// TIA Portal V15.1 export
// export: Created 2024-06-21T08:40:57.9475663Z, ExportSetting WithDefaults, DisplayName Totally Integrated Automation Portal, DisplayVersion V15.1 Update 5, DisplayName TIA Portal Openness, DisplayVersion V15.1 Update 5, DisplayName SINAMICS Startdrive Advanced, DisplayVersion V15.1, DisplayName G130, G150, S120, S150, SINAMICS MV, S210, DisplayVersion V15.1, DisplayName G110M, G120, G120C, G120D, G120P, DisplayVersion V15.1, DisplayName STEP 7 Professional, DisplayVersion V15.1 Update 5, DisplayName STEP 7 Safety, DisplayVersion V15.1, DisplayName WinCC Professional, DisplayVersion V15.1 Update 5, DisplayName SIMATIC Visualization Architect, DisplayVersion V15.1
FUNCTION_BLOCK "L10Alarm"   // FB1410, FBD
TITLE = L10Alarm
{ S7_Optimized_Access := 'FALSE' }
AUTHOR : VCC
FAMILY : AlarmHnd
NAME : 10Alarm
VERSION : 1.0
// ================================================================================
// This module is used everywhere 10 alarms has to be generated when one 
// (security) corresponding input becomes True.
// All alarms can be True only when the corresponding input Enable Alarm is also 
// True.
// When the conditions to generate the alarm is disappear, a boolean (one per 
// alarm) available to inform the upper level that the corresponding alarm can be 
// reset. All alarms are reset by means of the AlarmResetPB signal.
// ================================================================================
// stored: AutoNumber false, IsIECCheckEnabled false, SetENOAutomatically False, UDAEnableTagReadback false
   VAR_INPUT
      I_Input1 { ExternalAccessible := 'False'; ExternalVisible := 'False'; ExternalWritable := 'False'} : Bool;   // Input alarm 1
      I_AlarmClass1 { ExternalAccessible := 'False'; ExternalVisible := 'False'; ExternalWritable := 'False'} : Char;   // Alarm class -> A - B - C - D or E
      I_EnableAlarm1 { ExternalAccessible := 'False'; ExternalVisible := 'False'; ExternalWritable := 'False'} : Bool := TRUE;   // Enable alarm 1 from upper level
      I_Invisible1 { ExternalAccessible := 'False'; ExternalVisible := 'False'; ExternalWritable := 'False'} : Bool;   // Invisible 1
      I_Input2 { ExternalAccessible := 'False'; ExternalVisible := 'False'; ExternalWritable := 'False'} : Bool;   // Input alarm 2
      I_AlarmClass2 { ExternalAccessible := 'False'; ExternalVisible := 'False'; ExternalWritable := 'False'} : Char;   // Alarm class -> A - B - C - D or E
      I_EnableAlarm2 { ExternalAccessible := 'False'; ExternalVisible := 'False'; ExternalWritable := 'False'} : Bool := TRUE;   // Enable alarm 2 from upper level
      I_Invisible2 { ExternalAccessible := 'False'; ExternalVisible := 'False'; ExternalWritable := 'False'} : Bool;   // Invisible 2
      I_Input3 { ExternalAccessible := 'False'; ExternalVisible := 'False'; ExternalWritable := 'False'} : Bool;   // Input alarm 3
      I_AlarmClass3 { ExternalAccessible := 'False'; ExternalVisible := 'False'; ExternalWritable := 'False'} : Char;   // Alarm class -> A - B - C - D or E
      I_EnableAlarm3 { ExternalAccessible := 'False'; ExternalVisible := 'False'; ExternalWritable := 'False'} : Bool := TRUE;   // Enable alarm 3 from upper level
      I_Invisible3 { ExternalAccessible := 'False'; ExternalVisible := 'False'; ExternalWritable := 'False'} : Bool;   // Invisible 3
      I_Input4 { ExternalAccessible := 'False'; ExternalVisible := 'False'; ExternalWritable := 'False'} : Bool;   // Input alarm 4
      I_AlarmClass4 { ExternalAccessible := 'False'; ExternalVisible := 'False'; ExternalWritable := 'False'} : Char;   // Alarm class -> A - B - C - D or E
      I_EnableAlarm4 { ExternalAccessible := 'False'; ExternalVisible := 'False'; ExternalWritable := 'False'} : Bool := TRUE;   // Enable alarm 4 from upper level
      I_Invisible4 { ExternalAccessible := 'False'; ExternalVisible := 'False'; ExternalWritable := 'False'} : Bool;   // Invisible 4
      I_Input5 { ExternalAccessible := 'False'; ExternalVisible := 'False'; ExternalWritable := 'False'} : Bool;   // Input alarm 5
      I_AlarmClass5 { ExternalAccessible := 'False'; ExternalVisible := 'False'; ExternalWritable := 'False'} : Char;   // Alarm class -> A - B - C - D or E
      I_EnableAlarm5 { ExternalAccessible := 'False'; ExternalVisible := 'False'; ExternalWritable := 'False'} : Bool := TRUE;   // Enable alarm 5 from upper level
      I_Invisible5 { ExternalAccessible := 'False'; ExternalVisible := 'False'; ExternalWritable := 'False'} : Bool;   // Invisible 5
      I_Input6 { ExternalAccessible := 'False'; ExternalVisible := 'False'; ExternalWritable := 'False'} : Bool;   // Input alarm 6
      I_AlarmClass6 { ExternalAccessible := 'False'; ExternalVisible := 'False'; ExternalWritable := 'False'} : Char;   // Alarm class -> A - B - C - D or E
      I_EnableAlarm6 { ExternalAccessible := 'False'; ExternalVisible := 'False'; ExternalWritable := 'False'} : Bool := TRUE;   // Enable alarm 6 from upper level
      I_Invisible6 { ExternalAccessible := 'False'; ExternalVisible := 'False'; ExternalWritable := 'False'} : Bool;   // Invisible 6
      I_Input7 { ExternalAccessible := 'False'; ExternalVisible := 'False'; ExternalWritable := 'False'} : Bool;   // Input alarm 7
      I_AlarmClass7 { ExternalAccessible := 'False'; ExternalVisible := 'False'; ExternalWritable := 'False'} : Char;   // Alarm class -> A - B - C - D or E
      I_EnableAlarm7 { ExternalAccessible := 'False'; ExternalVisible := 'False'; ExternalWritable := 'False'} : Bool := TRUE;   // Enable alarm 7 from upper level
      I_Invisible7 { ExternalAccessible := 'False'; ExternalVisible := 'False'; ExternalWritable := 'False'} : Bool;   // Invisible 7
      I_Input8 { ExternalAccessible := 'False'; ExternalVisible := 'False'; ExternalWritable := 'False'} : Bool;   // Input alarm 8
      I_AlarmClass8 { ExternalAccessible := 'False'; ExternalVisible := 'False'; ExternalWritable := 'False'} : Char;   // Alarm class -> A - B - C - D or E
      I_EnableAlarm8 { ExternalAccessible := 'False'; ExternalVisible := 'False'; ExternalWritable := 'False'} : Bool := TRUE;   // Enable alarm 8 from upper level
      I_Invisible8 { ExternalAccessible := 'False'; ExternalVisible := 'False'; ExternalWritable := 'False'} : Bool;   // Invisible 8
      I_Input9 { ExternalAccessible := 'False'; ExternalVisible := 'False'; ExternalWritable := 'False'} : Bool;   // Input alarm 9 (normally open)
      I_AlarmClass9 { ExternalAccessible := 'False'; ExternalVisible := 'False'; ExternalWritable := 'False'} : Char;   // Alarm class -> A - B - C - D or E
      I_EnableAlarm9 { ExternalAccessible := 'False'; ExternalVisible := 'False'; ExternalWritable := 'False'} : Bool := TRUE;   // Enable alarm 9 from upper level
      I_Invisible9 { ExternalAccessible := 'False'; ExternalVisible := 'False'; ExternalWritable := 'False'} : Bool;   // Invisible 9
      I_Input10 { ExternalAccessible := 'False'; ExternalVisible := 'False'; ExternalWritable := 'False'} : Bool;   // Input alarm 10
      I_AlarmClass10 { ExternalAccessible := 'False'; ExternalVisible := 'False'; ExternalWritable := 'False'} : Char;   // Alarm class -> A - B - C - D or E
      I_EnableAlarm10 { ExternalAccessible := 'False'; ExternalVisible := 'False'; ExternalWritable := 'False'} : Bool := TRUE;   // Enable alarm 10 from upper level
      I_Invisible10 { ExternalAccessible := 'False'; ExternalVisible := 'False'; ExternalWritable := 'False'} : Bool;   // Invisible 10
      I_AlarmResetPB { ExternalAccessible := 'False'; ExternalVisible := 'False'; ExternalWritable := 'False'} : Bool;   // Alarm reset pushbutton is activated
   END_VAR
   VAR_OUTPUT
      O_Alarm1 { ExternalAccessible := 'False'; ExternalVisible := 'False'; ExternalWritable := 'False'} : Bool;   // Alarm 1
      O_Alarm2 { ExternalAccessible := 'False'; ExternalVisible := 'False'; ExternalWritable := 'False'} : Bool;   // Alarm 2
      O_Alarm3 { ExternalAccessible := 'False'; ExternalVisible := 'False'; ExternalWritable := 'False'} : Bool;   // Alarm 3
      O_Alarm4 { ExternalAccessible := 'False'; ExternalVisible := 'False'; ExternalWritable := 'False'} : Bool;   // Alarm 4
      O_Alarm5 { ExternalAccessible := 'False'; ExternalVisible := 'False'; ExternalWritable := 'False'} : Bool;   // Alarm 5
      O_Alarm6 { ExternalAccessible := 'False'; ExternalVisible := 'False'; ExternalWritable := 'False'} : Bool;   // Alarm 6
      O_Alarm7 { ExternalAccessible := 'False'; ExternalVisible := 'False'; ExternalWritable := 'False'} : Bool;   // Alarm 7
      O_Alarm8 { ExternalAccessible := 'False'; ExternalVisible := 'False'; ExternalWritable := 'False'} : Bool;   // Alarm 8
      O_Alarm9 { ExternalAccessible := 'False'; ExternalVisible := 'False'; ExternalWritable := 'False'} : Bool;   // Alarm 9
      O_Alarm10 { ExternalAccessible := 'False'; ExternalVisible := 'False'; ExternalWritable := 'False'} : Bool;   // Alarm 10
      O_AlarmABCondition { ExternalAccessible := 'False'; ExternalVisible := 'False'; ExternalWritable := 'False'} : Bool;   // Alarm AB condition
      H_IAnim1 { ExternalAccessible := 'False'; ExternalVisible := 'False'; ExternalWritable := 'False'} : Word;   // Icon Animation 1
      H_IAnim2 { ExternalAccessible := 'False'; ExternalVisible := 'False'; ExternalWritable := 'False'} : Word;   // Icon Animation 2
      H_IAnim3 { ExternalAccessible := 'False'; ExternalVisible := 'False'; ExternalWritable := 'False'} : Word;   // Icon Animation 3
      H_IAnim4 { ExternalAccessible := 'False'; ExternalVisible := 'False'; ExternalWritable := 'False'} : Word;   // Icon Animation 4
      H_IAnim5 { ExternalAccessible := 'False'; ExternalVisible := 'False'; ExternalWritable := 'False'} : Word;   // Icon Animation 5
      H_IAnim6 { ExternalAccessible := 'False'; ExternalVisible := 'False'; ExternalWritable := 'False'} : Word;   // Icon Animation 6
      H_IAnim7 { ExternalAccessible := 'False'; ExternalVisible := 'False'; ExternalWritable := 'False'} : Word;   // Icon Animation 7
      H_IAnim8 { ExternalAccessible := 'False'; ExternalVisible := 'False'; ExternalWritable := 'False'} : Word;   // Icon Animation 8
      H_IAnim9 { ExternalAccessible := 'False'; ExternalVisible := 'False'; ExternalWritable := 'False'} : Word;   // Icon Animation 9
      H_IAnim10 { ExternalAccessible := 'False'; ExternalVisible := 'False'; ExternalWritable := 'False'} : Word;   // Icon Animation 10
   END_VAR
   VAR DB_SPECIFIC
      H_Out : Struct   // HMI
         Anim1 : Word;   // HMI Animation of the object
         Anim2 : Word;   // HMI Animation of the object
         Anim3 : Word;   // HMI Animation of the object
         Anim4 : Word;   // HMI Animation of the object
         Anim5 : Word;   // HMI Animation of the object
         Anim6 : Word;   // HMI Animation of the object
         Anim7 : Word;   // HMI Animation of the object
         Anim8 : Word;   // HMI Animation of the object
         Anim9 : Word;   // HMI Animation of the object
         Anim10 : Word;   // HMI Animation of the object
         DBnr : Int;   // HMI Animation DB number
      END_STRUCT;
      Alarm1 { ExternalAccessible := 'False'; ExternalVisible := 'False'; ExternalWritable := 'False'} : Bool;   // Alarm 1
      AlarmClass1_A { ExternalAccessible := 'False'; ExternalVisible := 'False'; ExternalWritable := 'False'} : Bool;   // The alarm is from alarm class A
      AlarmClass1_B { ExternalAccessible := 'False'; ExternalVisible := 'False'; ExternalWritable := 'False'} : Bool;   // The alarm is from alarm class B
      AlarmClass1_C { ExternalAccessible := 'False'; ExternalVisible := 'False'; ExternalWritable := 'False'} : Bool;   // The alarm is from alarm class C
      AlarmClass1_D { ExternalAccessible := 'False'; ExternalVisible := 'False'; ExternalWritable := 'False'} : Bool;   // The alarm is from alarm class D
      AlarmClass1_E { ExternalAccessible := 'False'; ExternalVisible := 'False'; ExternalWritable := 'False'} : Bool;   // The alarm is from alarm class E
      Alarm1Cond { ExternalAccessible := 'False'; ExternalVisible := 'False'; ExternalWritable := 'False'} : Bool;   // Alarm 1 condition
      Alarm2 { ExternalAccessible := 'False'; ExternalVisible := 'False'; ExternalWritable := 'False'} : Bool;   // Alarm 2
      AlarmClass2_A { ExternalAccessible := 'False'; ExternalVisible := 'False'; ExternalWritable := 'False'} : Bool;   // The alarm is from alarm class A
      AlarmClass2_B { ExternalAccessible := 'False'; ExternalVisible := 'False'; ExternalWritable := 'False'} : Bool;   // The alarm is from alarm class B
      AlarmClass2_C { ExternalAccessible := 'False'; ExternalVisible := 'False'; ExternalWritable := 'False'} : Bool;   // The alarm is from alarm class C
      AlarmClass2_D { ExternalAccessible := 'False'; ExternalVisible := 'False'; ExternalWritable := 'False'} : Bool;   // The alarm is from alarm class D
      AlarmClass2_E { ExternalAccessible := 'False'; ExternalVisible := 'False'; ExternalWritable := 'False'} : Bool;   // The alarm is from alarm class E
      Alarm2Cond { ExternalAccessible := 'False'; ExternalVisible := 'False'; ExternalWritable := 'False'} : Bool;   // Alarm 2 condition
      Alarm3 { ExternalAccessible := 'False'; ExternalVisible := 'False'; ExternalWritable := 'False'} : Bool;   // Alarm 3
      AlarmClass3_A { ExternalAccessible := 'False'; ExternalVisible := 'False'; ExternalWritable := 'False'} : Bool;   // The alarm is from alarm class A
      AlarmClass3_B { ExternalAccessible := 'False'; ExternalVisible := 'False'; ExternalWritable := 'False'} : Bool;   // The alarm is from alarm class B
      AlarmClass3_C { ExternalAccessible := 'False'; ExternalVisible := 'False'; ExternalWritable := 'False'} : Bool;   // The alarm is from alarm class C
      AlarmClass3_D { ExternalAccessible := 'False'; ExternalVisible := 'False'; ExternalWritable := 'False'} : Bool;   // The alarm is from alarm class D
      AlarmClass3_E { ExternalAccessible := 'False'; ExternalVisible := 'False'; ExternalWritable := 'False'} : Bool;   // The alarm is from alarm class E
      Alarm3Cond { ExternalAccessible := 'False'; ExternalVisible := 'False'; ExternalWritable := 'False'} : Bool;   // Alarm 3 condition
      Alarm4 { ExternalAccessible := 'False'; ExternalVisible := 'False'; ExternalWritable := 'False'} : Bool;   // Alarm 4
      AlarmClass4_A { ExternalAccessible := 'False'; ExternalVisible := 'False'; ExternalWritable := 'False'} : Bool;   // The alarm is from alarm class A
      AlarmClass4_B { ExternalAccessible := 'False'; ExternalVisible := 'False'; ExternalWritable := 'False'} : Bool;   // The alarm is from alarm class B
      AlarmClass4_C { ExternalAccessible := 'False'; ExternalVisible := 'False'; ExternalWritable := 'False'} : Bool;   // The alarm is from alarm class C
      AlarmClass4_D { ExternalAccessible := 'False'; ExternalVisible := 'False'; ExternalWritable := 'False'} : Bool;   // The alarm is from alarm class D
      AlarmClass4_E { ExternalAccessible := 'False'; ExternalVisible := 'False'; ExternalWritable := 'False'} : Bool;   // The alarm is from alarm class E
      Alarm4Cond { ExternalAccessible := 'False'; ExternalVisible := 'False'; ExternalWritable := 'False'} : Bool;   // Alarm 4 condition
      Alarm5 { ExternalAccessible := 'False'; ExternalVisible := 'False'; ExternalWritable := 'False'} : Bool;   // Alarm 5
      AlarmClass5_A { ExternalAccessible := 'False'; ExternalVisible := 'False'; ExternalWritable := 'False'} : Bool;   // The alarm is from alarm class A
      AlarmClass5_B { ExternalAccessible := 'False'; ExternalVisible := 'False'; ExternalWritable := 'False'} : Bool;   // The alarm is from alarm class B
      AlarmClass5_C { ExternalAccessible := 'False'; ExternalVisible := 'False'; ExternalWritable := 'False'} : Bool;   // The alarm is from alarm class C
      AlarmClass5_D { ExternalAccessible := 'False'; ExternalVisible := 'False'; ExternalWritable := 'False'} : Bool;   // The alarm is from alarm class D
      AlarmClass5_E { ExternalAccessible := 'False'; ExternalVisible := 'False'; ExternalWritable := 'False'} : Bool;   // The alarm is from alarm class E
      Alarm5Cond { ExternalAccessible := 'False'; ExternalVisible := 'False'; ExternalWritable := 'False'} : Bool;   // Alarm 5 condition
      Alarm6 { ExternalAccessible := 'False'; ExternalVisible := 'False'; ExternalWritable := 'False'} : Bool;   // Alarm 6
      AlarmClass6_A { ExternalAccessible := 'False'; ExternalVisible := 'False'; ExternalWritable := 'False'} : Bool;   // The alarm is from alarm class A
      AlarmClass6_B { ExternalAccessible := 'False'; ExternalVisible := 'False'; ExternalWritable := 'False'} : Bool;   // The alarm is from alarm class B
      AlarmClass6_C { ExternalAccessible := 'False'; ExternalVisible := 'False'; ExternalWritable := 'False'} : Bool;   // The alarm is from alarm class C
      AlarmClass6_D { ExternalAccessible := 'False'; ExternalVisible := 'False'; ExternalWritable := 'False'} : Bool;   // The alarm is from alarm class D
      AlarmClass6_E { ExternalAccessible := 'False'; ExternalVisible := 'False'; ExternalWritable := 'False'} : Bool;   // The alarm is from alarm class E
      Alarm6Cond { ExternalAccessible := 'False'; ExternalVisible := 'False'; ExternalWritable := 'False'} : Bool;   // Alarm 6 condition
      Alarm7 { ExternalAccessible := 'False'; ExternalVisible := 'False'; ExternalWritable := 'False'} : Bool;   // Alarm 7
      AlarmClass7_A { ExternalAccessible := 'False'; ExternalVisible := 'False'; ExternalWritable := 'False'} : Bool;   // The alarm is from alarm class A
      AlarmClass7_B { ExternalAccessible := 'False'; ExternalVisible := 'False'; ExternalWritable := 'False'} : Bool;   // The alarm is from alarm class B
      AlarmClass7_C { ExternalAccessible := 'False'; ExternalVisible := 'False'; ExternalWritable := 'False'} : Bool;   // The alarm is from alarm class C
      AlarmClass7_D { ExternalAccessible := 'False'; ExternalVisible := 'False'; ExternalWritable := 'False'} : Bool;   // The alarm is from alarm class D
      AlarmClass7_E { ExternalAccessible := 'False'; ExternalVisible := 'False'; ExternalWritable := 'False'} : Bool;   // The alarm is from alarm class E
      Alarm7Cond { ExternalAccessible := 'False'; ExternalVisible := 'False'; ExternalWritable := 'False'} : Bool;   // Alarm 7 condition
      Alarm8 { ExternalAccessible := 'False'; ExternalVisible := 'False'; ExternalWritable := 'False'} : Bool;   // Alarm 8
      AlarmClass8_A { ExternalAccessible := 'False'; ExternalVisible := 'False'; ExternalWritable := 'False'} : Bool;   // The alarm is from alarm class A
      AlarmClass8_B { ExternalAccessible := 'False'; ExternalVisible := 'False'; ExternalWritable := 'False'} : Bool;   // The alarm is from alarm class B
      AlarmClass8_C { ExternalAccessible := 'False'; ExternalVisible := 'False'; ExternalWritable := 'False'} : Bool;   // The alarm is from alarm class C
      AlarmClass8_D { ExternalAccessible := 'False'; ExternalVisible := 'False'; ExternalWritable := 'False'} : Bool;   // The alarm is from alarm class D
      AlarmClass8_E { ExternalAccessible := 'False'; ExternalVisible := 'False'; ExternalWritable := 'False'} : Bool;   // The alarm is from alarm class E
      Alarm8Cond { ExternalAccessible := 'False'; ExternalVisible := 'False'; ExternalWritable := 'False'} : Bool;   // Alarm 8 condition
      Alarm9 { ExternalAccessible := 'False'; ExternalVisible := 'False'; ExternalWritable := 'False'} : Bool;   // Alarm 9
      AlarmClass9_A { ExternalAccessible := 'False'; ExternalVisible := 'False'; ExternalWritable := 'False'} : Bool;   // The alarm is from alarm class A
      AlarmClass9_B { ExternalAccessible := 'False'; ExternalVisible := 'False'; ExternalWritable := 'False'} : Bool;   // The alarm is from alarm class B
      AlarmClass9_C { ExternalAccessible := 'False'; ExternalVisible := 'False'; ExternalWritable := 'False'} : Bool;   // The alarm is from alarm class C
      AlarmClass9_D { ExternalAccessible := 'False'; ExternalVisible := 'False'; ExternalWritable := 'False'} : Bool;   // The alarm is from alarm class D
      AlarmClass9_E { ExternalAccessible := 'False'; ExternalVisible := 'False'; ExternalWritable := 'False'} : Bool;   // The alarm is from alarm class E
      Alarm9Cond { ExternalAccessible := 'False'; ExternalVisible := 'False'; ExternalWritable := 'False'} : Bool;   // Alarm 9 condition
      Alarm10 { ExternalAccessible := 'False'; ExternalVisible := 'False'; ExternalWritable := 'False'} : Bool;   // Alarm 10
      AlarmClass10_A { ExternalAccessible := 'False'; ExternalVisible := 'False'; ExternalWritable := 'False'} : Bool;   // The alarm is from alarm class A
      AlarmClass10_B { ExternalAccessible := 'False'; ExternalVisible := 'False'; ExternalWritable := 'False'} : Bool;   // The alarm is from alarm class B
      AlarmClass10_C { ExternalAccessible := 'False'; ExternalVisible := 'False'; ExternalWritable := 'False'} : Bool;   // The alarm is from alarm class C
      AlarmClass10_D { ExternalAccessible := 'False'; ExternalVisible := 'False'; ExternalWritable := 'False'} : Bool;   // The alarm is from alarm class D
      AlarmClass10_E { ExternalAccessible := 'False'; ExternalVisible := 'False'; ExternalWritable := 'False'} : Bool;   // The alarm is from alarm class E
      Alarm10Cond { ExternalAccessible := 'False'; ExternalVisible := 'False'; ExternalWritable := 'False'} : Bool;   // Alarm 10 condition
      DBnr { ExternalAccessible := 'False'; ExternalVisible := 'False'; ExternalWritable := 'False'} : Int;   // HMI DB number
   END_VAR
BEGIN

NETWORK
TITLE = **** 1 - Inputs **** DB number
// DB number
      L     DINO;
      T     #DBnr;

NETWORK
TITLE = **** 1 - Inputs **** Alarm class 1
// Alarm class
// Alarm class = E
      L     #I_AlarmClass1;
      L     'E';
      ==I;
      =     #AlarmClass1_E;

// Alarm class = D
      L     #I_AlarmClass1;
      L     'D';
      ==I;
      =     #AlarmClass1_D;

// Alarm class = C
      L     #I_AlarmClass1;
      L     'C';
      ==I;
      =     #AlarmClass1_C;

// Alarm class = B
      L     #I_AlarmClass1;
      L     'B';
      ==I;
      =     #AlarmClass1_B;

// Alarm class = A
      AN    #AlarmClass1_B;
      AN    #AlarmClass1_C;
      AN    #AlarmClass1_D;
      AN    #AlarmClass1_E;
      =     #AlarmClass1_A;


NETWORK
TITLE = **** 1 - Inputs **** Alarm class 2
// Alarm class
// Alarm class = E
      L     #I_AlarmClass2;
      L     'E';
      ==I;
      =     #AlarmClass2_E;

// Alarm class = D
      L     #I_AlarmClass2;
      L     'D';
      ==I;
      =     #AlarmClass2_D;

// Alarm class = C
      L     #I_AlarmClass2;
      L     'C';
      ==I;
      =     #AlarmClass2_C;

// Alarm class = B
      L     #I_AlarmClass2;
      L     'B';
      ==I;
      =     #AlarmClass2_B;

// Alarm class = A
      AN    #AlarmClass2_B;
      AN    #AlarmClass2_C;
      AN    #AlarmClass2_D;
      AN    #AlarmClass2_E;
      =     #AlarmClass2_A;


NETWORK
TITLE = **** 1 - Inputs **** Alarm class 3
// Alarm class
// Alarm class = E
      L     #I_AlarmClass3;
      L     'E';
      ==I;
      =     #AlarmClass3_E;

// Alarm class = D
      L     #I_AlarmClass3;
      L     'D';
      ==I;
      =     #AlarmClass3_D;

// Alarm class = C
      L     #I_AlarmClass3;
      L     'C';
      ==I;
      =     #AlarmClass3_C;

// Alarm class = B
      L     #I_AlarmClass3;
      L     'B';
      ==I;
      =     #AlarmClass3_B;

// Alarm class = A
      AN    #AlarmClass3_B;
      AN    #AlarmClass3_C;
      AN    #AlarmClass3_D;
      AN    #AlarmClass3_E;
      =     #AlarmClass3_A;


NETWORK
TITLE = **** 1 - Inputs **** Alarm class 4
// Alarm class
// Alarm class = E
      L     #I_AlarmClass4;
      L     'E';
      ==I;
      =     #AlarmClass4_E;

// Alarm class = D
      L     #I_AlarmClass4;
      L     'D';
      ==I;
      =     #AlarmClass4_D;

// Alarm class = C
      L     #I_AlarmClass4;
      L     'C';
      ==I;
      =     #AlarmClass4_C;

// Alarm class = B
      L     #I_AlarmClass4;
      L     'B';
      ==I;
      =     #AlarmClass4_B;

// Alarm class = A
      AN    #AlarmClass4_B;
      AN    #AlarmClass4_C;
      AN    #AlarmClass4_D;
      AN    #AlarmClass4_E;
      =     #AlarmClass4_A;


NETWORK
TITLE = **** 1 - Inputs **** Alarm class 5
// Alarm class
// Alarm class = E
      L     #I_AlarmClass5;
      L     'E';
      ==I;
      =     #AlarmClass5_E;

// Alarm class = D
      L     #I_AlarmClass5;
      L     'D';
      ==I;
      =     #AlarmClass5_D;

// Alarm class = C
      L     #I_AlarmClass5;
      L     'C';
      ==I;
      =     #AlarmClass5_C;

// Alarm class = B
      L     #I_AlarmClass5;
      L     'B';
      ==I;
      =     #AlarmClass5_B;

// Alarm class = A
      AN    #AlarmClass5_B;
      AN    #AlarmClass5_C;
      AN    #AlarmClass5_D;
      AN    #AlarmClass5_E;
      =     #AlarmClass5_A;


NETWORK
TITLE = **** 1 - Inputs **** Alarm class 6
// Alarm class
// Alarm class = E
      L     #I_AlarmClass6;
      L     'E';
      ==I;
      =     #AlarmClass6_E;

// Alarm class = D
      L     #I_AlarmClass6;
      L     'D';
      ==I;
      =     #AlarmClass6_D;

// Alarm class = C
      L     #I_AlarmClass6;
      L     'C';
      ==I;
      =     #AlarmClass6_C;

// Alarm class = B
      L     #I_AlarmClass6;
      L     'B';
      ==I;
      =     #AlarmClass6_B;

// Alarm class = A
      AN    #AlarmClass6_B;
      AN    #AlarmClass6_C;
      AN    #AlarmClass6_D;
      AN    #AlarmClass6_E;
      =     #AlarmClass6_A;


NETWORK
TITLE = **** 1 - Inputs **** Alarm class 7
// Alarm class
// Alarm class = E
      L     #I_AlarmClass7;
      L     'E';
      ==I;
      =     #AlarmClass7_E;

// Alarm class = D
      L     #I_AlarmClass7;
      L     'D';
      ==I;
      =     #AlarmClass7_D;

// Alarm class = C
      L     #I_AlarmClass7;
      L     'C';
      ==I;
      =     #AlarmClass7_C;

// Alarm class = B
      L     #I_AlarmClass7;
      L     'B';
      ==I;
      =     #AlarmClass7_B;

// Alarm class = A
      AN    #AlarmClass7_B;
      AN    #AlarmClass7_C;
      AN    #AlarmClass7_D;
      AN    #AlarmClass7_E;
      =     #AlarmClass7_A;


NETWORK
TITLE = **** 1 - Inputs **** Alarm class 8
// Alarm class
// Alarm class = E
      L     #I_AlarmClass8;
      L     'E';
      ==I;
      =     #AlarmClass8_E;

// Alarm class = D
      L     #I_AlarmClass8;
      L     'D';
      ==I;
      =     #AlarmClass8_D;

// Alarm class = C
      L     #I_AlarmClass8;
      L     'C';
      ==I;
      =     #AlarmClass8_C;

// Alarm class = B
      L     #I_AlarmClass8;
      L     'B';
      ==I;
      =     #AlarmClass8_B;

// Alarm class = A
      AN    #AlarmClass8_B;
      AN    #AlarmClass8_C;
      AN    #AlarmClass8_D;
      AN    #AlarmClass8_E;
      =     #AlarmClass8_A;


NETWORK
TITLE = **** 1 - Inputs **** Alarm class 9
// Alarm class
// Alarm class = E
      L     #I_AlarmClass9;
      L     'E';
      ==I;
      =     #AlarmClass9_E;

// Alarm class = D
      L     #I_AlarmClass9;
      L     'D';
      ==I;
      =     #AlarmClass9_D;

// Alarm class = C
      L     #I_AlarmClass9;
      L     'C';
      ==I;
      =     #AlarmClass9_C;

// Alarm class = B
      L     #I_AlarmClass9;
      L     'B';
      ==I;
      =     #AlarmClass9_B;

// Alarm class = A
      AN    #AlarmClass9_B;
      AN    #AlarmClass9_C;
      AN    #AlarmClass9_D;
      AN    #AlarmClass9_E;
      =     #AlarmClass9_A;


NETWORK
TITLE = **** 1 - Inputs **** Alarm class 10
// Alarm class
// Alarm class = E
      L     #I_AlarmClass10;
      L     'E';
      ==I;
      =     #AlarmClass10_E;

// Alarm class = D
      L     #I_AlarmClass10;
      L     'D';
      ==I;
      =     #AlarmClass10_D;

// Alarm class = C
      L     #I_AlarmClass10;
      L     'C';
      ==I;
      =     #AlarmClass10_C;

// Alarm class = B
      L     #I_AlarmClass10;
      L     'B';
      ==I;
      =     #AlarmClass10_B;

// Alarm class = A
      AN    #AlarmClass10_B;
      AN    #AlarmClass10_C;
      AN    #AlarmClass10_D;
      AN    #AlarmClass10_E;
      =     #AlarmClass10_A;


REGION Network 12: **** 2.2 - Alarms - Alarms Generation **** Alarm Condition 1
   // Condition for Alarm 1
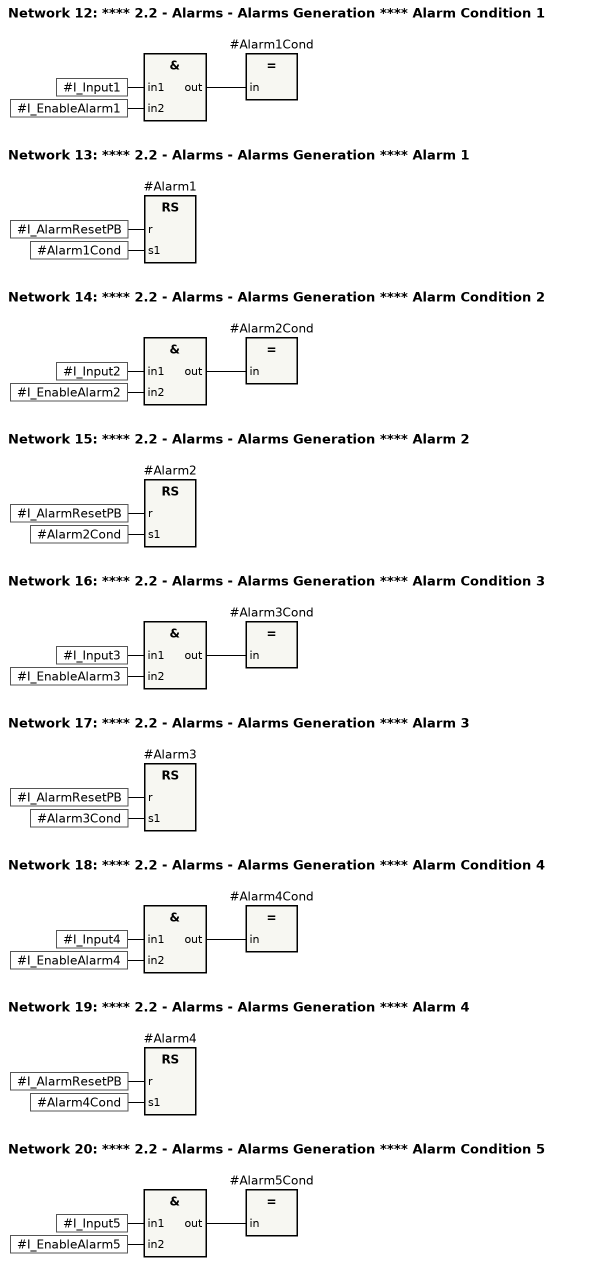
   #Alarm1Cond := #I_Input1 AND #I_EnableAlarm1;
END_REGION

REGION Network 13: **** 2.2 - Alarms - Alarms Generation **** Alarm 1
   // Creation of the Alarm 1
   IF #I_AlarmResetPB THEN
       #Alarm1 := FALSE;   // RS flip-flop
   END_IF;
   IF #Alarm1Cond THEN #Alarm1 := TRUE; END_IF;
END_REGION

REGION Network 14: **** 2.2 - Alarms - Alarms Generation **** Alarm Condition 2
   // Condition for Alarm 2
   #Alarm2Cond := #I_Input2 AND #I_EnableAlarm2;
END_REGION

REGION Network 15: **** 2.2 - Alarms - Alarms Generation **** Alarm 2
   // Creation of the Alarm 2
   IF #I_AlarmResetPB THEN
       #Alarm2 := FALSE;   // RS flip-flop
   END_IF;
   IF #Alarm2Cond THEN #Alarm2 := TRUE; END_IF;
END_REGION

REGION Network 16: **** 2.2 - Alarms - Alarms Generation **** Alarm Condition 3
   // Condition for Alarm 3
   #Alarm3Cond := #I_Input3 AND #I_EnableAlarm3;
END_REGION

REGION Network 17: **** 2.2 - Alarms - Alarms Generation **** Alarm 3
   // Creation of the Alarm 3
   IF #I_AlarmResetPB THEN
       #Alarm3 := FALSE;   // RS flip-flop
   END_IF;
   IF #Alarm3Cond THEN #Alarm3 := TRUE; END_IF;
END_REGION

REGION Network 18: **** 2.2 - Alarms - Alarms Generation **** Alarm Condition 4
   // Condition for Alarm 4
   #Alarm4Cond := #I_Input4 AND #I_EnableAlarm4;
END_REGION

REGION Network 19: **** 2.2 - Alarms - Alarms Generation **** Alarm 4
   // Creation of the Alarm 4
   IF #I_AlarmResetPB THEN
       #Alarm4 := FALSE;   // RS flip-flop
   END_IF;
   IF #Alarm4Cond THEN #Alarm4 := TRUE; END_IF;
END_REGION

REGION Network 20: **** 2.2 - Alarms - Alarms Generation **** Alarm Condition 5
   // Condition for Alarm 5
   #Alarm5Cond := #I_Input5 AND #I_EnableAlarm5;
END_REGION

REGION Network 21: **** 2.2 - Alarms - Alarms Generation **** Alarm 5
   // Creation of the Alarm 5
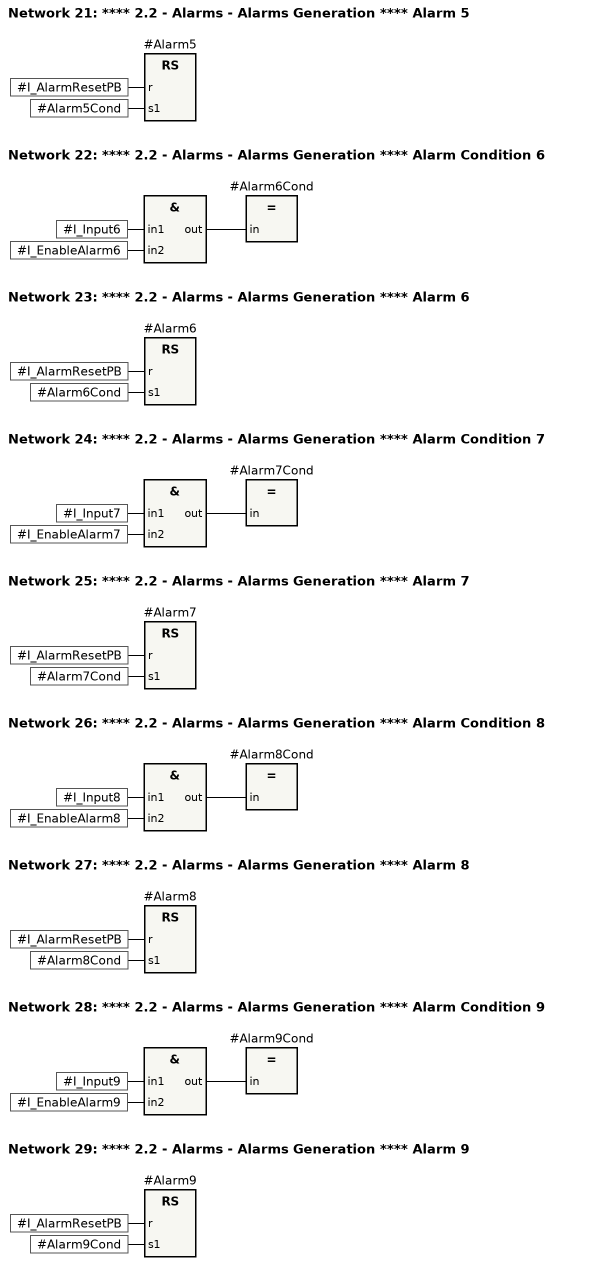
   IF #I_AlarmResetPB THEN
       #Alarm5 := FALSE;   // RS flip-flop
   END_IF;
   IF #Alarm5Cond THEN #Alarm5 := TRUE; END_IF;
END_REGION

REGION Network 22: **** 2.2 - Alarms - Alarms Generation **** Alarm Condition 6
   // Condition for Alarm 6
   #Alarm6Cond := #I_Input6 AND #I_EnableAlarm6;
END_REGION

REGION Network 23: **** 2.2 - Alarms - Alarms Generation **** Alarm 6
   // Creation of the Alarm 6
   IF #I_AlarmResetPB THEN
       #Alarm6 := FALSE;   // RS flip-flop
   END_IF;
   IF #Alarm6Cond THEN #Alarm6 := TRUE; END_IF;
END_REGION

REGION Network 24: **** 2.2 - Alarms - Alarms Generation **** Alarm Condition 7
   // Condition for Alarm 7
   #Alarm7Cond := #I_Input7 AND #I_EnableAlarm7;
END_REGION

REGION Network 25: **** 2.2 - Alarms - Alarms Generation **** Alarm 7
   // Creation of the Alarm 7
   IF #I_AlarmResetPB THEN
       #Alarm7 := FALSE;   // RS flip-flop
   END_IF;
   IF #Alarm7Cond THEN #Alarm7 := TRUE; END_IF;
END_REGION

REGION Network 26: **** 2.2 - Alarms - Alarms Generation **** Alarm Condition 8
   // Condition for Alarm 8
   #Alarm8Cond := #I_Input8 AND #I_EnableAlarm8;
END_REGION

REGION Network 27: **** 2.2 - Alarms - Alarms Generation **** Alarm 8
   // Creation of the Alarm 8
   IF #I_AlarmResetPB THEN
       #Alarm8 := FALSE;   // RS flip-flop
   END_IF;
   IF #Alarm8Cond THEN #Alarm8 := TRUE; END_IF;
END_REGION

REGION Network 28: **** 2.2 - Alarms - Alarms Generation **** Alarm Condition 9
   // Condition for Alarm 9
   #Alarm9Cond := #I_Input9 AND #I_EnableAlarm9;
END_REGION

REGION Network 29: **** 2.2 - Alarms - Alarms Generation **** Alarm 9
   // Creation of the Alarm 9
   IF #I_AlarmResetPB THEN
       #Alarm9 := FALSE;   // RS flip-flop
   END_IF;
   IF #Alarm9Cond THEN #Alarm9 := TRUE; END_IF;
END_REGION

REGION Network 30: **** 2.2 - Alarms - Alarms Generation **** Alarm Condition 10
   // Condition for Alarm 10
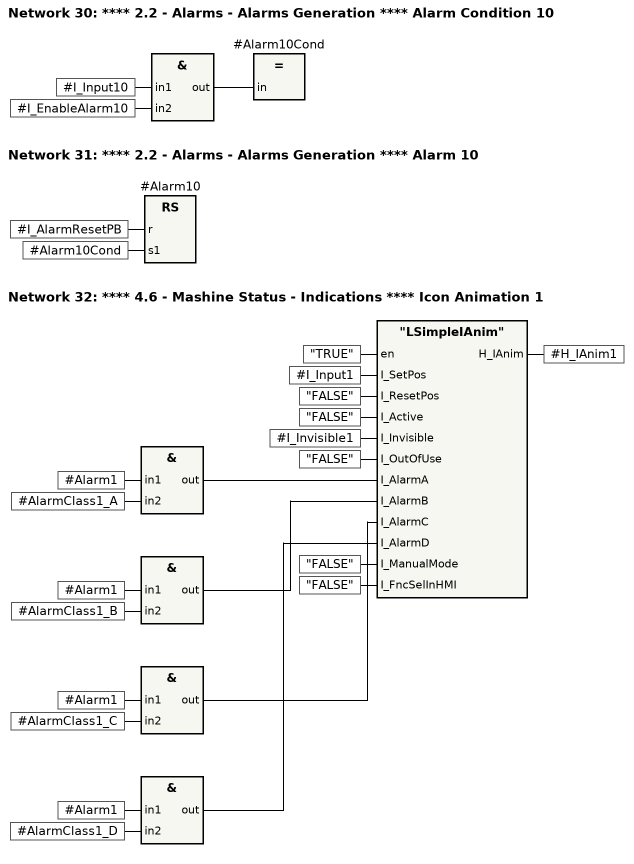
   #Alarm10Cond := #I_Input10 AND #I_EnableAlarm10;
END_REGION

REGION Network 31: **** 2.2 - Alarms - Alarms Generation **** Alarm 10
   // Creation of the Alarm 10
   IF #I_AlarmResetPB THEN
       #Alarm10 := FALSE;   // RS flip-flop
   END_IF;
   IF #Alarm10Cond THEN #Alarm10 := TRUE; END_IF;
END_REGION

REGION Network 32: **** 4.6 - Mashine Status - Indications **** Icon Animation 1
   // Icon Animation 1
   IF "TRUE" THEN
       "LSimpleIAnim"(I_SetPos := #I_Input1,
                      I_ResetPos := "FALSE",
                      I_Active := "FALSE",
                      I_Invisible := #I_Invisible1,
                      I_OutOfUse := "FALSE",
                      I_AlarmA := #Alarm1 AND #AlarmClass1_A,
                      I_AlarmB := #Alarm1 AND #AlarmClass1_B,
                      I_AlarmC := #Alarm1 AND #AlarmClass1_C,
                      I_AlarmD := #Alarm1 AND #AlarmClass1_D,
                      I_ManualMode := "FALSE",
                      I_FncSelInHMI := "FALSE",
                      H_IAnim => #H_IAnim1);
   END_IF;
END_REGION

REGION Network 33: **** 4.6 - Mashine Status - Indications **** Icon Animation 2
   // Icon Animation 2
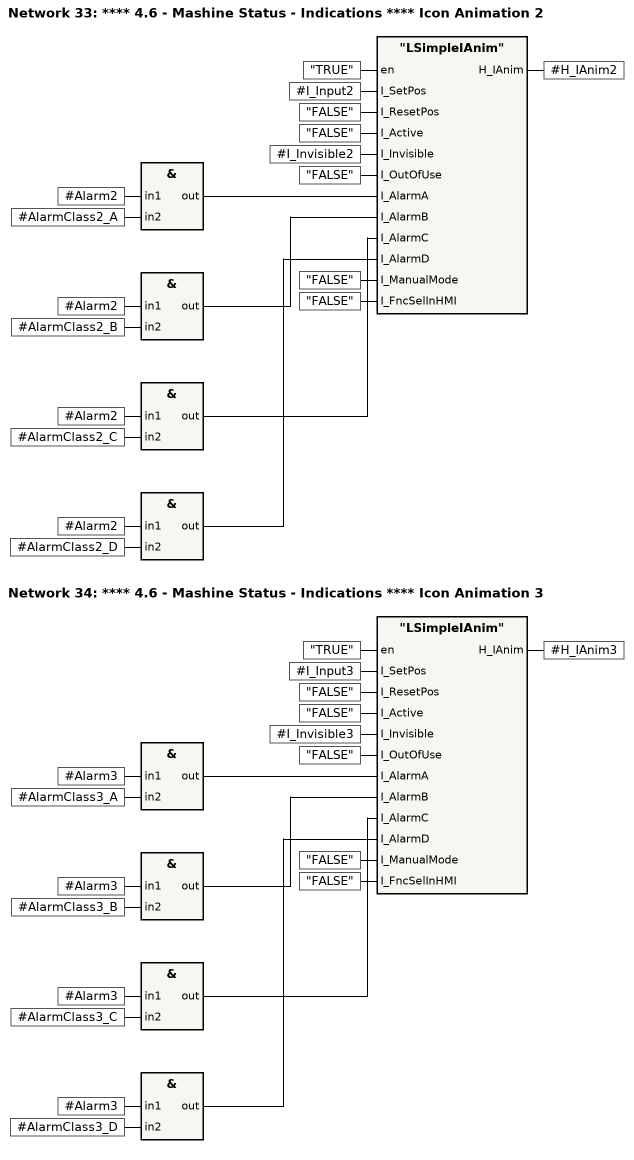
   IF "TRUE" THEN
       "LSimpleIAnim"(I_SetPos := #I_Input2,
                      I_ResetPos := "FALSE",
                      I_Active := "FALSE",
                      I_Invisible := #I_Invisible2,
                      I_OutOfUse := "FALSE",
                      I_AlarmA := #Alarm2 AND #AlarmClass2_A,
                      I_AlarmB := #Alarm2 AND #AlarmClass2_B,
                      I_AlarmC := #Alarm2 AND #AlarmClass2_C,
                      I_AlarmD := #Alarm2 AND #AlarmClass2_D,
                      I_ManualMode := "FALSE",
                      I_FncSelInHMI := "FALSE",
                      H_IAnim => #H_IAnim2);
   END_IF;
END_REGION

REGION Network 34: **** 4.6 - Mashine Status - Indications **** Icon Animation 3
   // Icon Animation 3
   IF "TRUE" THEN
       "LSimpleIAnim"(I_SetPos := #I_Input3,
                      I_ResetPos := "FALSE",
                      I_Active := "FALSE",
                      I_Invisible := #I_Invisible3,
                      I_OutOfUse := "FALSE",
                      I_AlarmA := #Alarm3 AND #AlarmClass3_A,
                      I_AlarmB := #Alarm3 AND #AlarmClass3_B,
                      I_AlarmC := #Alarm3 AND #AlarmClass3_C,
                      I_AlarmD := #Alarm3 AND #AlarmClass3_D,
                      I_ManualMode := "FALSE",
                      I_FncSelInHMI := "FALSE",
                      H_IAnim => #H_IAnim3);
   END_IF;
END_REGION

REGION Network 35: **** 4.6 - Mashine Status - Indications **** Icon Animation 4
   // Icon Animation 4
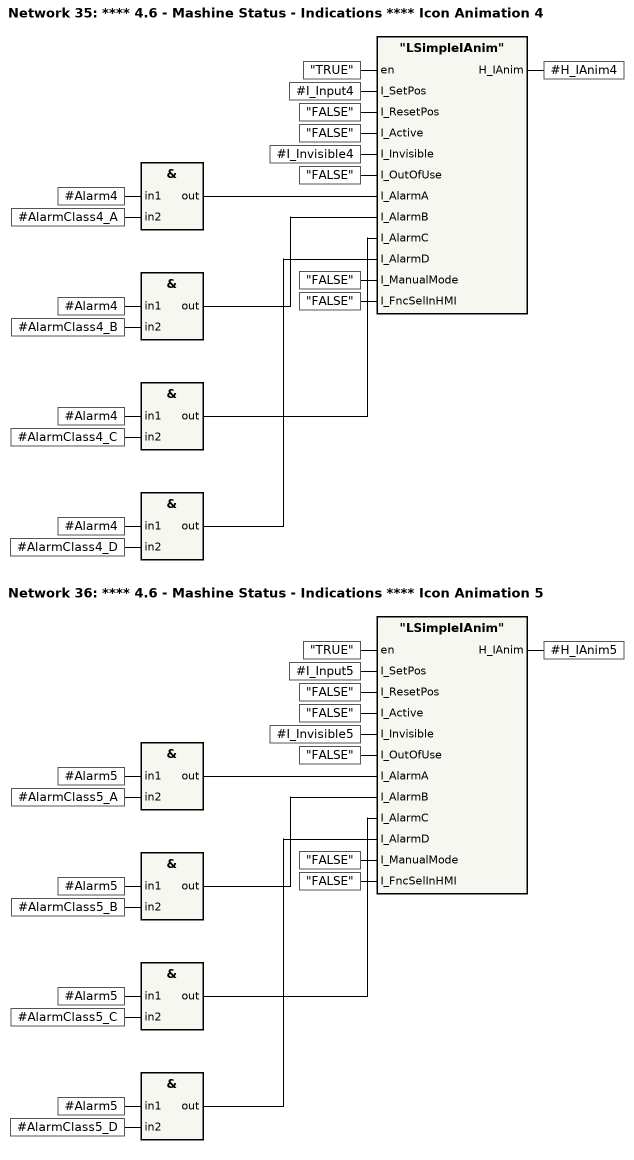
   IF "TRUE" THEN
       "LSimpleIAnim"(I_SetPos := #I_Input4,
                      I_ResetPos := "FALSE",
                      I_Active := "FALSE",
                      I_Invisible := #I_Invisible4,
                      I_OutOfUse := "FALSE",
                      I_AlarmA := #Alarm4 AND #AlarmClass4_A,
                      I_AlarmB := #Alarm4 AND #AlarmClass4_B,
                      I_AlarmC := #Alarm4 AND #AlarmClass4_C,
                      I_AlarmD := #Alarm4 AND #AlarmClass4_D,
                      I_ManualMode := "FALSE",
                      I_FncSelInHMI := "FALSE",
                      H_IAnim => #H_IAnim4);
   END_IF;
END_REGION

REGION Network 36: **** 4.6 - Mashine Status - Indications **** Icon Animation 5
   // Icon Animation 5
   IF "TRUE" THEN
       "LSimpleIAnim"(I_SetPos := #I_Input5,
                      I_ResetPos := "FALSE",
                      I_Active := "FALSE",
                      I_Invisible := #I_Invisible5,
                      I_OutOfUse := "FALSE",
                      I_AlarmA := #Alarm5 AND #AlarmClass5_A,
                      I_AlarmB := #Alarm5 AND #AlarmClass5_B,
                      I_AlarmC := #Alarm5 AND #AlarmClass5_C,
                      I_AlarmD := #Alarm5 AND #AlarmClass5_D,
                      I_ManualMode := "FALSE",
                      I_FncSelInHMI := "FALSE",
                      H_IAnim => #H_IAnim5);
   END_IF;
END_REGION

REGION Network 37: **** 4.6 - Mashine Status - Indications **** Icon Animation 6
   // Icon Animation 6
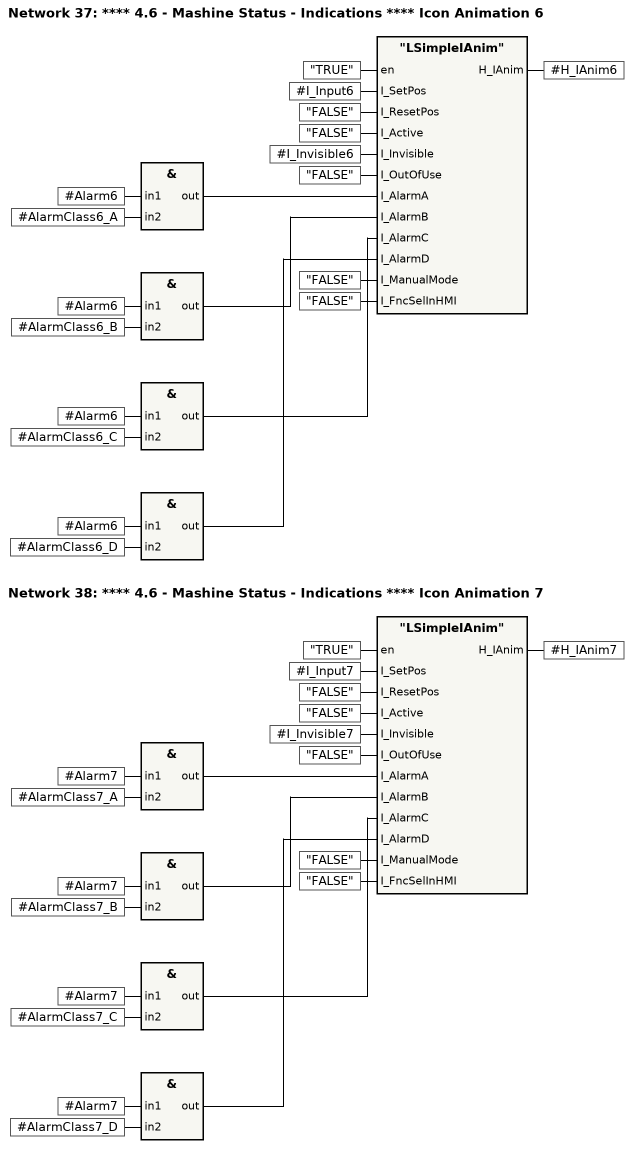
   IF "TRUE" THEN
       "LSimpleIAnim"(I_SetPos := #I_Input6,
                      I_ResetPos := "FALSE",
                      I_Active := "FALSE",
                      I_Invisible := #I_Invisible6,
                      I_OutOfUse := "FALSE",
                      I_AlarmA := #Alarm6 AND #AlarmClass6_A,
                      I_AlarmB := #Alarm6 AND #AlarmClass6_B,
                      I_AlarmC := #Alarm6 AND #AlarmClass6_C,
                      I_AlarmD := #Alarm6 AND #AlarmClass6_D,
                      I_ManualMode := "FALSE",
                      I_FncSelInHMI := "FALSE",
                      H_IAnim => #H_IAnim6);
   END_IF;
END_REGION

REGION Network 38: **** 4.6 - Mashine Status - Indications **** Icon Animation 7
   // Icon Animation 7
   IF "TRUE" THEN
       "LSimpleIAnim"(I_SetPos := #I_Input7,
                      I_ResetPos := "FALSE",
                      I_Active := "FALSE",
                      I_Invisible := #I_Invisible7,
                      I_OutOfUse := "FALSE",
                      I_AlarmA := #Alarm7 AND #AlarmClass7_A,
                      I_AlarmB := #Alarm7 AND #AlarmClass7_B,
                      I_AlarmC := #Alarm7 AND #AlarmClass7_C,
                      I_AlarmD := #Alarm7 AND #AlarmClass7_D,
                      I_ManualMode := "FALSE",
                      I_FncSelInHMI := "FALSE",
                      H_IAnim => #H_IAnim7);
   END_IF;
END_REGION

REGION Network 39: **** 4.6 - Mashine Status - Indications **** Icon Animation 8
   // Icon Animation 8
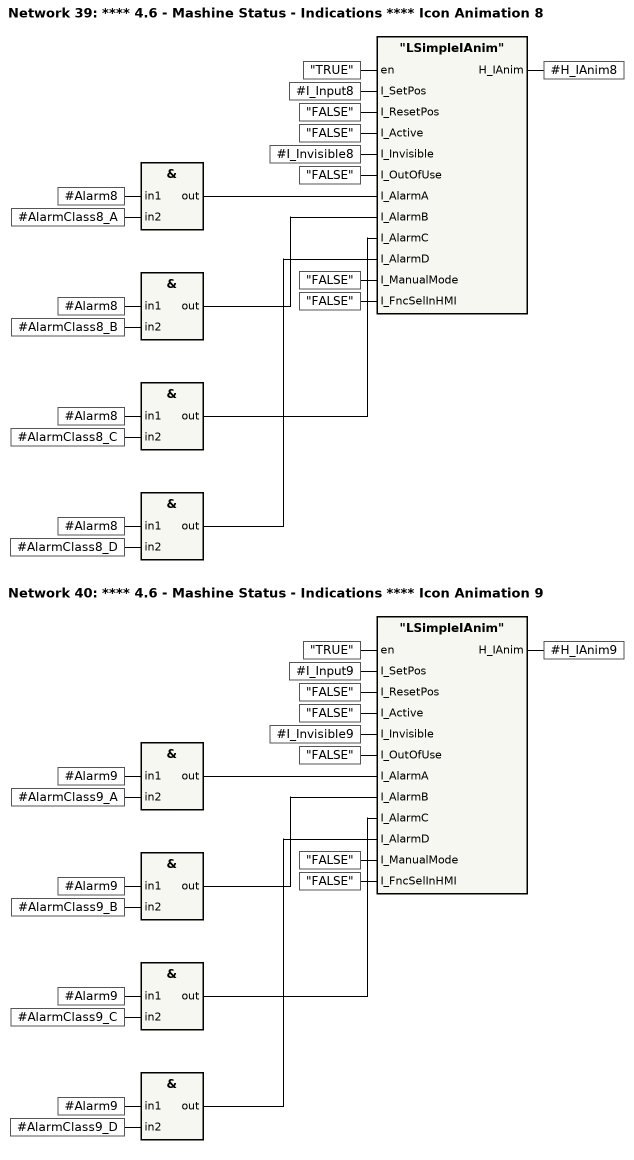
   IF "TRUE" THEN
       "LSimpleIAnim"(I_SetPos := #I_Input8,
                      I_ResetPos := "FALSE",
                      I_Active := "FALSE",
                      I_Invisible := #I_Invisible8,
                      I_OutOfUse := "FALSE",
                      I_AlarmA := #Alarm8 AND #AlarmClass8_A,
                      I_AlarmB := #Alarm8 AND #AlarmClass8_B,
                      I_AlarmC := #Alarm8 AND #AlarmClass8_C,
                      I_AlarmD := #Alarm8 AND #AlarmClass8_D,
                      I_ManualMode := "FALSE",
                      I_FncSelInHMI := "FALSE",
                      H_IAnim => #H_IAnim8);
   END_IF;
END_REGION

REGION Network 40: **** 4.6 - Mashine Status - Indications **** Icon Animation 9
   // Icon Animation 9
   IF "TRUE" THEN
       "LSimpleIAnim"(I_SetPos := #I_Input9,
                      I_ResetPos := "FALSE",
                      I_Active := "FALSE",
                      I_Invisible := #I_Invisible9,
                      I_OutOfUse := "FALSE",
                      I_AlarmA := #Alarm9 AND #AlarmClass9_A,
                      I_AlarmB := #Alarm9 AND #AlarmClass9_B,
                      I_AlarmC := #Alarm9 AND #AlarmClass9_C,
                      I_AlarmD := #Alarm9 AND #AlarmClass9_D,
                      I_ManualMode := "FALSE",
                      I_FncSelInHMI := "FALSE",
                      H_IAnim => #H_IAnim9);
   END_IF;
END_REGION

REGION Network 41: **** 4.6 - Mashine Status - Indications **** Icon Animation 10
   // Icon Animation 10
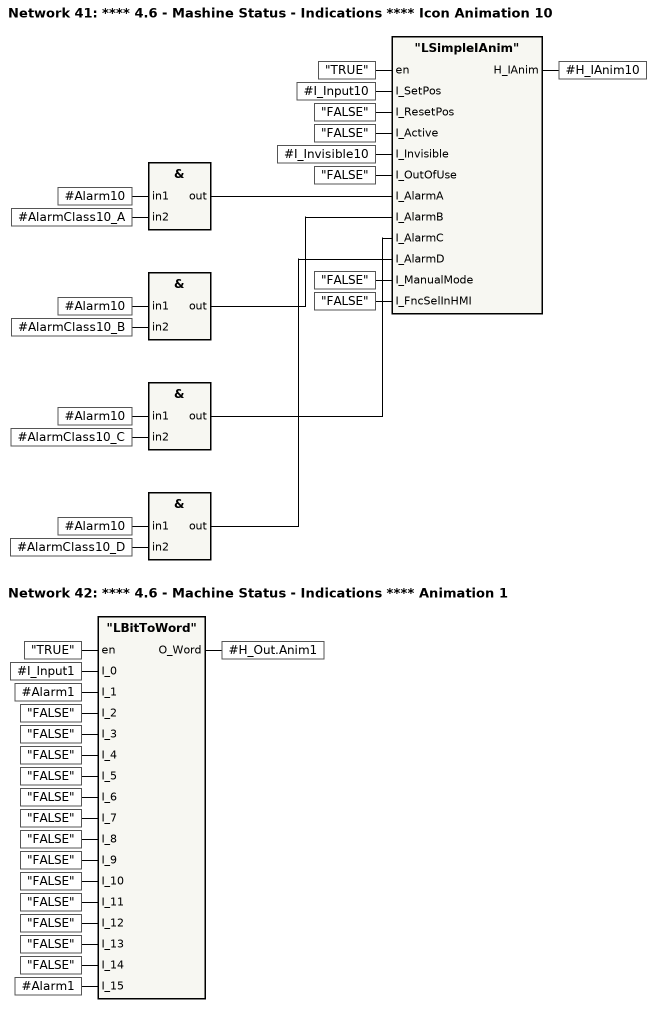
   IF "TRUE" THEN
       "LSimpleIAnim"(I_SetPos := #I_Input10,
                      I_ResetPos := "FALSE",
                      I_Active := "FALSE",
                      I_Invisible := #I_Invisible10,
                      I_OutOfUse := "FALSE",
                      I_AlarmA := #Alarm10 AND #AlarmClass10_A,
                      I_AlarmB := #Alarm10 AND #AlarmClass10_B,
                      I_AlarmC := #Alarm10 AND #AlarmClass10_C,
                      I_AlarmD := #Alarm10 AND #AlarmClass10_D,
                      I_ManualMode := "FALSE",
                      I_FncSelInHMI := "FALSE",
                      H_IAnim => #H_IAnim10);
   END_IF;
END_REGION

REGION Network 42: **** 4.6 - Machine Status - Indications **** Animation 1
   // Animation 1
   IF "TRUE" THEN
       "LBitToWord"(I_0 := #I_Input1,
                    I_1 := #Alarm1,
                    I_2 := "FALSE",
                    I_3 := "FALSE",
                    I_4 := "FALSE",
                    I_5 := "FALSE",
                    I_6 := "FALSE",
                    I_7 := "FALSE",
                    I_8 := "FALSE",
                    I_9 := "FALSE",
                    I_10 := "FALSE",
                    I_11 := "FALSE",
                    I_12 := "FALSE",
                    I_13 := "FALSE",
                    I_14 := "FALSE",
                    I_15 := #Alarm1,
                    O_Word => #H_Out.Anim1);
   END_IF;
END_REGION

REGION Network 43: **** 4.6 - Machine Status - Indications **** Animation 2
   // Animation 2
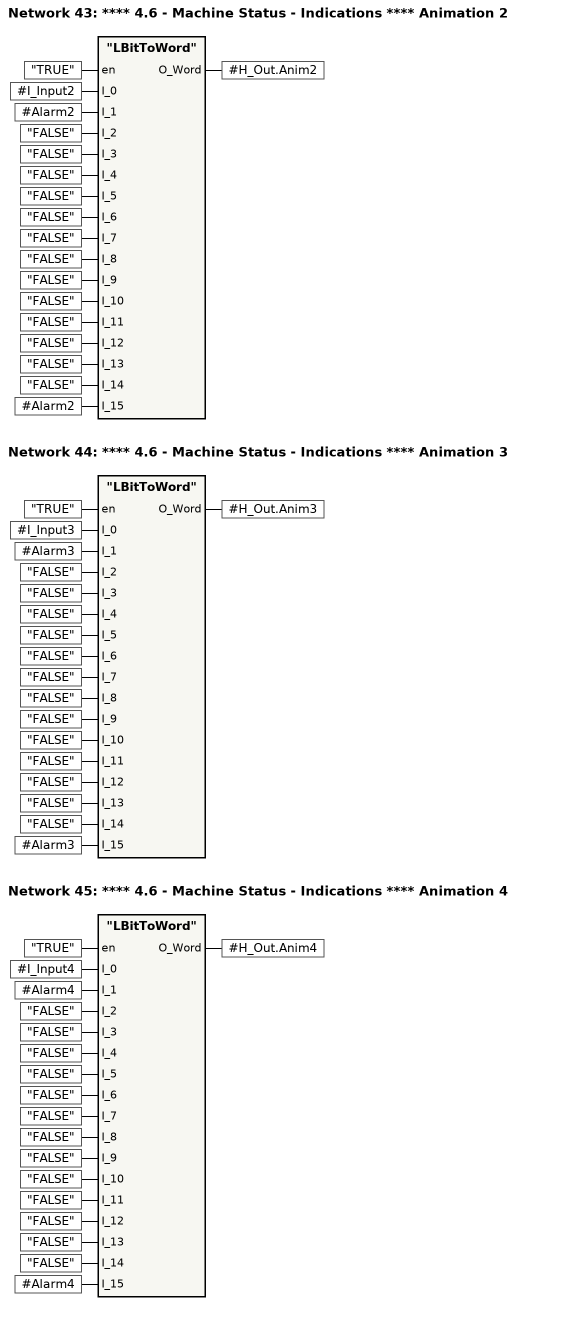
   IF "TRUE" THEN
       "LBitToWord"(I_0 := #I_Input2,
                    I_1 := #Alarm2,
                    I_2 := "FALSE",
                    I_3 := "FALSE",
                    I_4 := "FALSE",
                    I_5 := "FALSE",
                    I_6 := "FALSE",
                    I_7 := "FALSE",
                    I_8 := "FALSE",
                    I_9 := "FALSE",
                    I_10 := "FALSE",
                    I_11 := "FALSE",
                    I_12 := "FALSE",
                    I_13 := "FALSE",
                    I_14 := "FALSE",
                    I_15 := #Alarm2,
                    O_Word => #H_Out.Anim2);
   END_IF;
END_REGION

REGION Network 44: **** 4.6 - Machine Status - Indications **** Animation 3
   // Animation 3
   IF "TRUE" THEN
       "LBitToWord"(I_0 := #I_Input3,
                    I_1 := #Alarm3,
                    I_2 := "FALSE",
                    I_3 := "FALSE",
                    I_4 := "FALSE",
                    I_5 := "FALSE",
                    I_6 := "FALSE",
                    I_7 := "FALSE",
                    I_8 := "FALSE",
                    I_9 := "FALSE",
                    I_10 := "FALSE",
                    I_11 := "FALSE",
                    I_12 := "FALSE",
                    I_13 := "FALSE",
                    I_14 := "FALSE",
                    I_15 := #Alarm3,
                    O_Word => #H_Out.Anim3);
   END_IF;
END_REGION

REGION Network 45: **** 4.6 - Machine Status - Indications **** Animation 4
   // Animation 4
   IF "TRUE" THEN
       "LBitToWord"(I_0 := #I_Input4,
                    I_1 := #Alarm4,
                    I_2 := "FALSE",
                    I_3 := "FALSE",
                    I_4 := "FALSE",
                    I_5 := "FALSE",
                    I_6 := "FALSE",
                    I_7 := "FALSE",
                    I_8 := "FALSE",
                    I_9 := "FALSE",
                    I_10 := "FALSE",
                    I_11 := "FALSE",
                    I_12 := "FALSE",
                    I_13 := "FALSE",
                    I_14 := "FALSE",
                    I_15 := #Alarm4,
                    O_Word => #H_Out.Anim4);
   END_IF;
END_REGION

REGION Network 46: **** 4.6 - Machine Status - Indications **** Animation 5
   // Animation 5
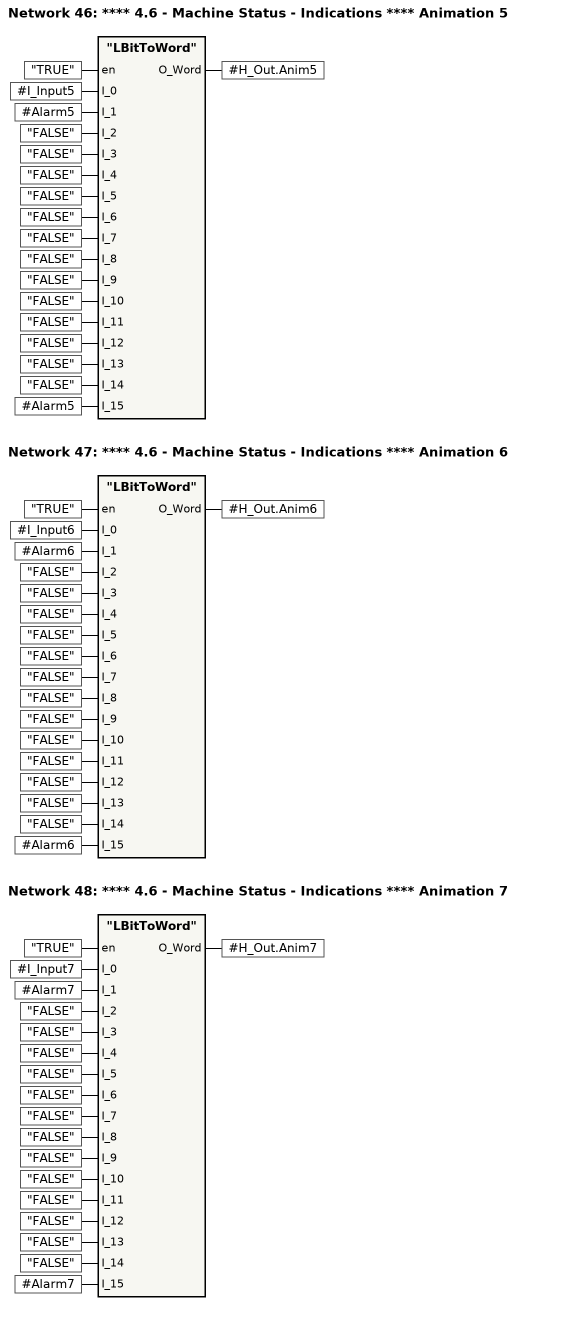
   IF "TRUE" THEN
       "LBitToWord"(I_0 := #I_Input5,
                    I_1 := #Alarm5,
                    I_2 := "FALSE",
                    I_3 := "FALSE",
                    I_4 := "FALSE",
                    I_5 := "FALSE",
                    I_6 := "FALSE",
                    I_7 := "FALSE",
                    I_8 := "FALSE",
                    I_9 := "FALSE",
                    I_10 := "FALSE",
                    I_11 := "FALSE",
                    I_12 := "FALSE",
                    I_13 := "FALSE",
                    I_14 := "FALSE",
                    I_15 := #Alarm5,
                    O_Word => #H_Out.Anim5);
   END_IF;
END_REGION

REGION Network 47: **** 4.6 - Machine Status - Indications **** Animation 6
   // Animation 6
   IF "TRUE" THEN
       "LBitToWord"(I_0 := #I_Input6,
                    I_1 := #Alarm6,
                    I_2 := "FALSE",
                    I_3 := "FALSE",
                    I_4 := "FALSE",
                    I_5 := "FALSE",
                    I_6 := "FALSE",
                    I_7 := "FALSE",
                    I_8 := "FALSE",
                    I_9 := "FALSE",
                    I_10 := "FALSE",
                    I_11 := "FALSE",
                    I_12 := "FALSE",
                    I_13 := "FALSE",
                    I_14 := "FALSE",
                    I_15 := #Alarm6,
                    O_Word => #H_Out.Anim6);
   END_IF;
END_REGION

REGION Network 48: **** 4.6 - Machine Status - Indications **** Animation 7
   // Animation 7
   IF "TRUE" THEN
       "LBitToWord"(I_0 := #I_Input7,
                    I_1 := #Alarm7,
                    I_2 := "FALSE",
                    I_3 := "FALSE",
                    I_4 := "FALSE",
                    I_5 := "FALSE",
                    I_6 := "FALSE",
                    I_7 := "FALSE",
                    I_8 := "FALSE",
                    I_9 := "FALSE",
                    I_10 := "FALSE",
                    I_11 := "FALSE",
                    I_12 := "FALSE",
                    I_13 := "FALSE",
                    I_14 := "FALSE",
                    I_15 := #Alarm7,
                    O_Word => #H_Out.Anim7);
   END_IF;
END_REGION

REGION Network 49: **** 4.6 - Machine Status - Indications **** Animation 8
   // Animation 8
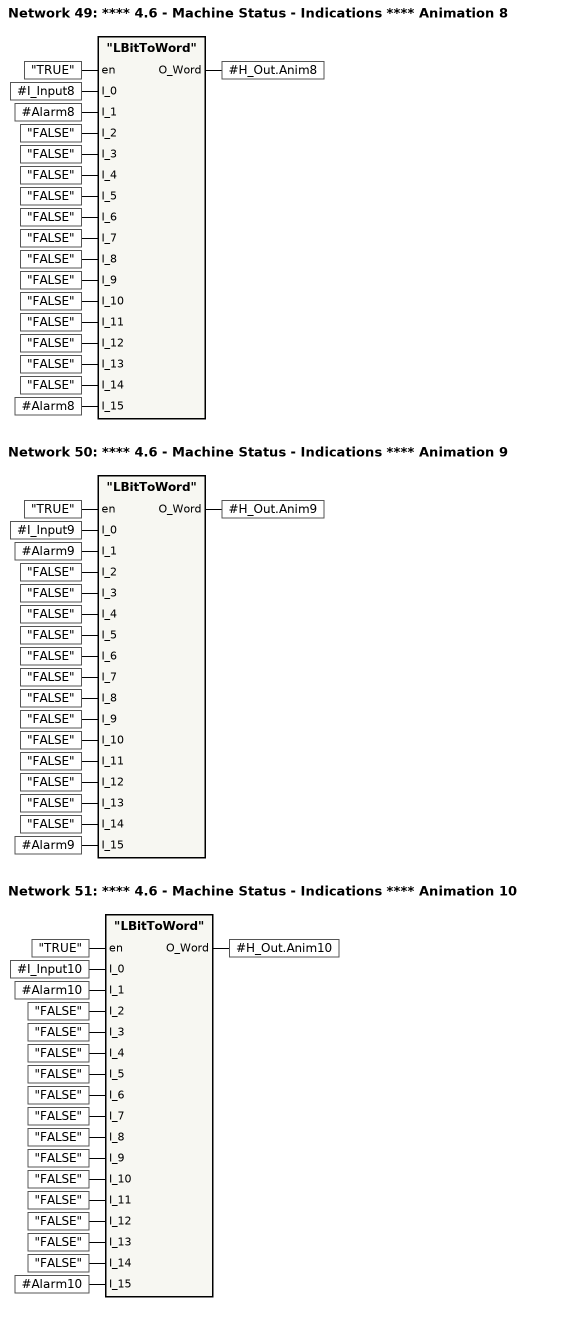
   IF "TRUE" THEN
       "LBitToWord"(I_0 := #I_Input8,
                    I_1 := #Alarm8,
                    I_2 := "FALSE",
                    I_3 := "FALSE",
                    I_4 := "FALSE",
                    I_5 := "FALSE",
                    I_6 := "FALSE",
                    I_7 := "FALSE",
                    I_8 := "FALSE",
                    I_9 := "FALSE",
                    I_10 := "FALSE",
                    I_11 := "FALSE",
                    I_12 := "FALSE",
                    I_13 := "FALSE",
                    I_14 := "FALSE",
                    I_15 := #Alarm8,
                    O_Word => #H_Out.Anim8);
   END_IF;
END_REGION

REGION Network 50: **** 4.6 - Machine Status - Indications **** Animation 9
   // Animation 9
   IF "TRUE" THEN
       "LBitToWord"(I_0 := #I_Input9,
                    I_1 := #Alarm9,
                    I_2 := "FALSE",
                    I_3 := "FALSE",
                    I_4 := "FALSE",
                    I_5 := "FALSE",
                    I_6 := "FALSE",
                    I_7 := "FALSE",
                    I_8 := "FALSE",
                    I_9 := "FALSE",
                    I_10 := "FALSE",
                    I_11 := "FALSE",
                    I_12 := "FALSE",
                    I_13 := "FALSE",
                    I_14 := "FALSE",
                    I_15 := #Alarm9,
                    O_Word => #H_Out.Anim9);
   END_IF;
END_REGION

REGION Network 51: **** 4.6 - Machine Status - Indications **** Animation 10
   // Animation 10
   IF "TRUE" THEN
       "LBitToWord"(I_0 := #I_Input10,
                    I_1 := #Alarm10,
                    I_2 := "FALSE",
                    I_3 := "FALSE",
                    I_4 := "FALSE",
                    I_5 := "FALSE",
                    I_6 := "FALSE",
                    I_7 := "FALSE",
                    I_8 := "FALSE",
                    I_9 := "FALSE",
                    I_10 := "FALSE",
                    I_11 := "FALSE",
                    I_12 := "FALSE",
                    I_13 := "FALSE",
                    I_14 := "FALSE",
                    I_15 := #Alarm10,
                    O_Word => #H_Out.Anim10);
   END_IF;
END_REGION

REGION Network 52: **** 4.6 - Machine status - Indications **** Animation DB number
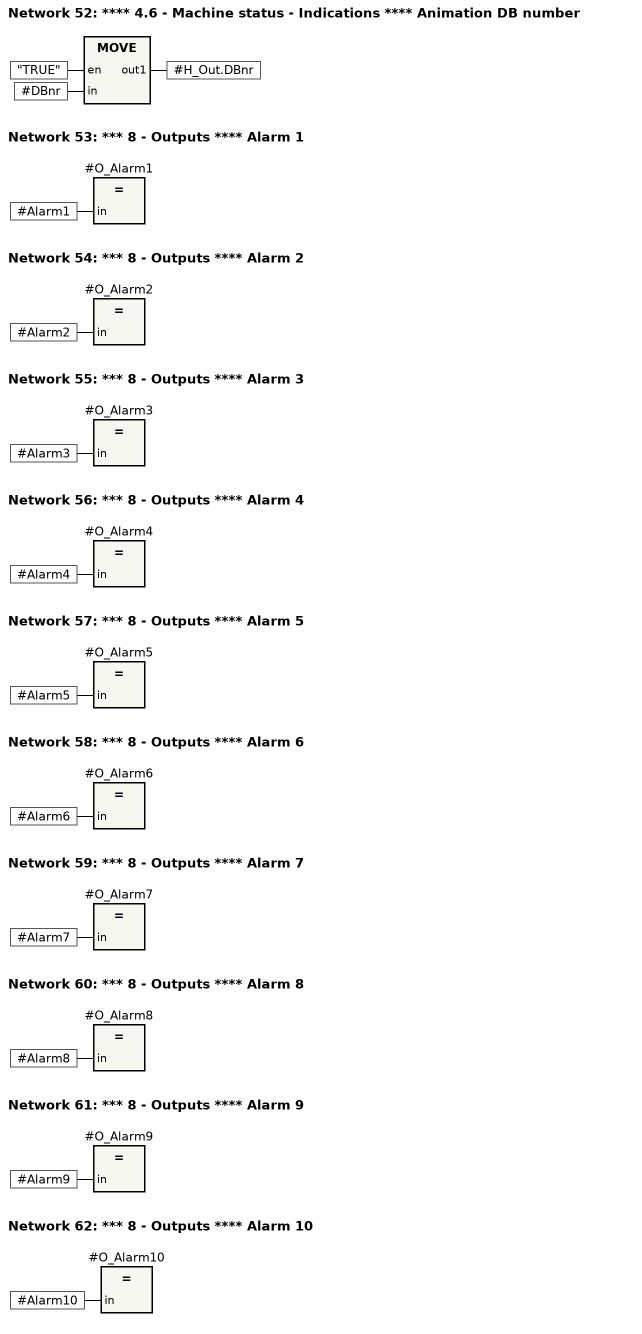
   IF "TRUE" THEN #H_Out.DBnr := #DBnr; END_IF;
END_REGION

REGION Network 53: *** 8 - Outputs **** Alarm 1
   // Output of the Alarm 1
   #O_Alarm1 := #Alarm1;
END_REGION

REGION Network 54: *** 8 - Outputs **** Alarm 2
   // Output of the Alarm 2
   #O_Alarm2 := #Alarm2;
END_REGION

REGION Network 55: *** 8 - Outputs **** Alarm 3
   // Output of the Alarm 3
   #O_Alarm3 := #Alarm3;
END_REGION

REGION Network 56: *** 8 - Outputs **** Alarm 4
   // Output of the Alarm 4
   #O_Alarm4 := #Alarm4;
END_REGION

REGION Network 57: *** 8 - Outputs **** Alarm 5
   // Output of the Alarm 5
   #O_Alarm5 := #Alarm5;
END_REGION

REGION Network 58: *** 8 - Outputs **** Alarm 6
   // Output of the Alarm 6
   #O_Alarm6 := #Alarm6;
END_REGION

REGION Network 59: *** 8 - Outputs **** Alarm 7
   // Output of the Alarm 7
   #O_Alarm7 := #Alarm7;
END_REGION

REGION Network 60: *** 8 - Outputs **** Alarm 8
   // Output of the Alarm 8
   #O_Alarm8 := #Alarm8;
END_REGION

REGION Network 61: *** 8 - Outputs **** Alarm 9
   // Output of the Alarm 9
   #O_Alarm9 := #Alarm9;
END_REGION

REGION Network 62: *** 8 - Outputs **** Alarm 10
   // Output of the Alarm 10
   #O_Alarm10 := #Alarm10;
END_REGION

REGION Network 63: **** 8 - Outputs **** Alarm AB Condition
   // Alarm AB condition
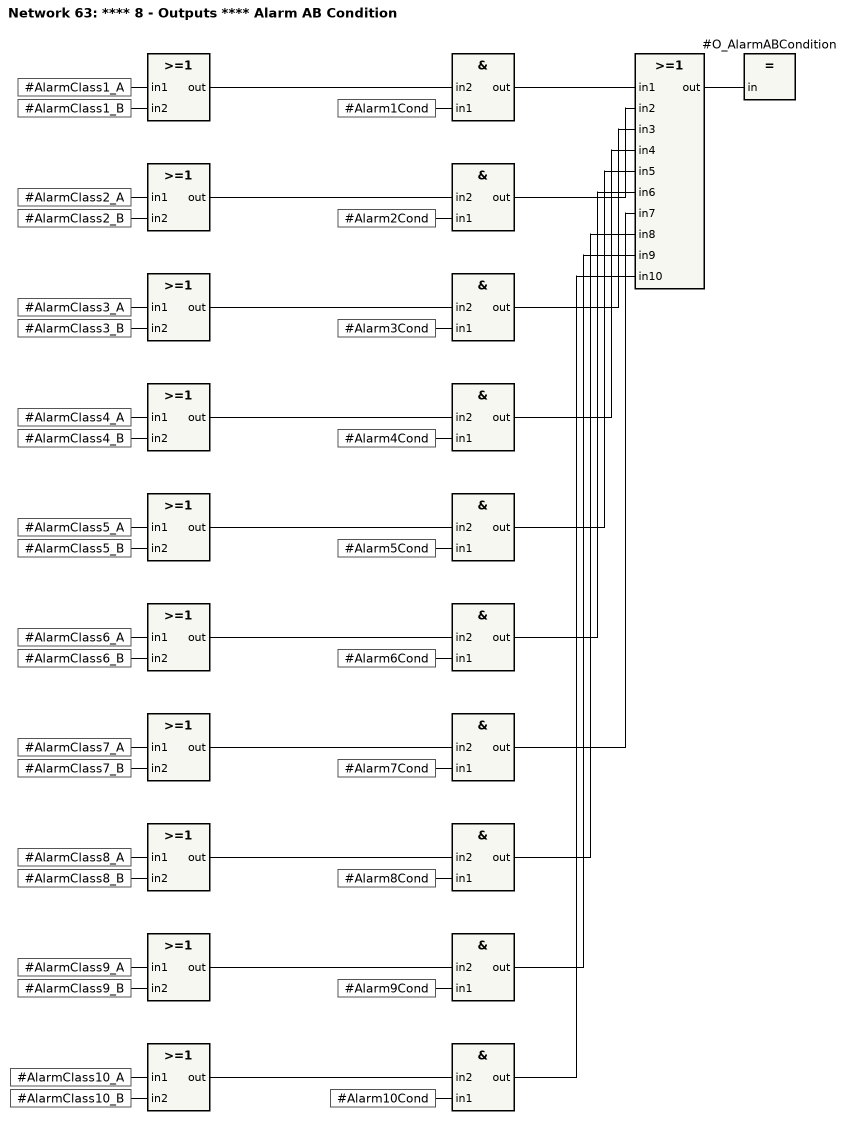
   #O_AlarmABCondition := ((#AlarmClass1_A OR #AlarmClass1_B) AND #Alarm1Cond) OR ((#AlarmClass2_A OR #AlarmClass2_B) AND #Alarm2Cond) OR ((#AlarmClass3_A OR #AlarmClass3_B) AND #Alarm3Cond) OR ((#AlarmClass4_A OR #AlarmClass4_B) AND #Alarm4Cond) OR ((#AlarmClass5_A OR #AlarmClass5_B) AND #Alarm5Cond) OR ((#AlarmClass6_A OR #AlarmClass6_B) AND #Alarm6Cond) OR ((#AlarmClass7_A OR #AlarmClass7_B) AND #Alarm7Cond) OR ((#AlarmClass8_A OR #AlarmClass8_B) AND #Alarm8Cond) OR ((#AlarmClass9_A OR #AlarmClass9_B) AND #Alarm9Cond) OR ((#AlarmClass10_A OR #AlarmClass10_B) AND #Alarm10Cond);
END_REGION
END_FUNCTION_BLOCK
